// TIA Portal V21 export
FUNCTION "DIG IP" : Void   // FC3, LAD
{ S7_Optimized_Access := 'TRUE' }
// stored: SetENOAutomatically false
   VAR_TEMP   // added for the SCL form of the ladder/FBD networks
      _w1 : Bool;
      _w2 : Bool;
      _w3 : Bool;
      _w4 : Bool;
      _w5 : Bool;
   END_VAR
BEGIN

REGION Network 1: BLOCK CALL
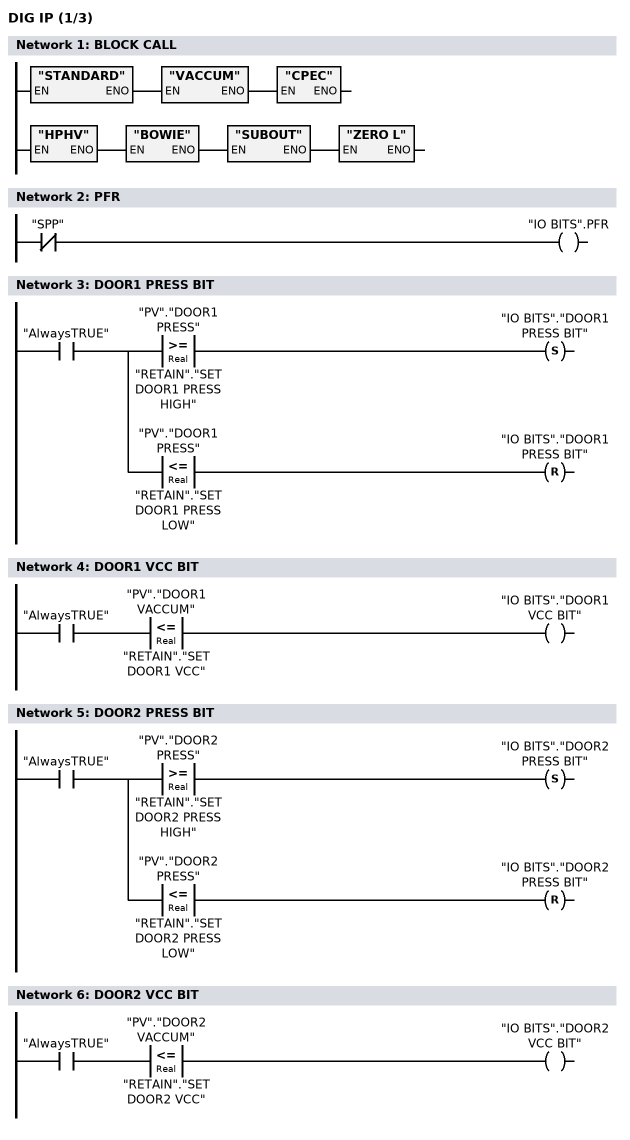
   RUNG wire#powerrail
      "STANDARD"()
      "VACCUM"()
      "CPEC"()
   END_RUNG
   RUNG wire#powerrail
      "HPHV"()
      "BOWIE"()
      "SUBOUT"()
      "ZERO L"()
   END_RUNG
   // the same network as SCL:
   "STANDARD"(ENO => #_w1);
   "VACCUM"(EN := #_w1, ENO => #_w2);
   IF #_w2 THEN "CPEC"(); END_IF;
   "HPHV"(ENO => #_w3);
   "BOWIE"(EN := #_w3, ENO => #_w4);
   "SUBOUT"(EN := #_w4, ENO => #_w5);
   IF #_w5 THEN "ZERO L"(); END_IF;
END_REGION

REGION Network 2: PFR
   RUNG wire#powerrail
      I_Contact( "SPP" )
      Coil( "IO BITS".PFR )
   END_RUNG
   // the same network as SCL:
   "IO BITS".PFR := NOT "SPP";
END_REGION

REGION Network 3: DOOR1 PRESS BIT
   RUNG wire#powerrail
      Contact( "AlwaysTRUE" )
      wire#w1
      { S7_Templates := "SrcType := Real" } GE_Contact(in1 := "PV"."DOOR1 PRESS", in2 := "RETAIN"."SET DOOR1 PRESS HIGH")
      S_Coil( "IO BITS"."DOOR1 PRESS BIT" )
   END_RUNG
   RUNG wire#w1
      { S7_Templates := "SrcType := Real" } LE_Contact(in1 := "PV"."DOOR1 PRESS", in2 := "RETAIN"."SET DOOR1 PRESS LOW")
      R_Coil( "IO BITS"."DOOR1 PRESS BIT" )
   END_RUNG
   // the same network as SCL:
   IF "AlwaysTRUE" AND ("PV"."DOOR1 PRESS" >= "RETAIN"."SET DOOR1 PRESS HIGH") THEN
       "IO BITS"."DOOR1 PRESS BIT" := TRUE;
   END_IF;
   IF "AlwaysTRUE" AND ("PV"."DOOR1 PRESS" <= "RETAIN"."SET DOOR1 PRESS LOW") THEN
       "IO BITS"."DOOR1 PRESS BIT" := FALSE;
   END_IF;
END_REGION

REGION Network 4: DOOR1 VCC BIT
   RUNG wire#powerrail
      Contact( "AlwaysTRUE" )
      { S7_Templates := "SrcType := Real" } LE_Contact(in1 := "PV"."DOOR1 VACCUM", in2 := "RETAIN"."SET DOOR1 VCC")
      Coil( "IO BITS"."DOOR1 VCC BIT" )
   END_RUNG
   // the same network as SCL:
   "IO BITS"."DOOR1 VCC BIT" := "AlwaysTRUE" AND ("PV"."DOOR1 VACCUM" <= "RETAIN"."SET DOOR1 VCC");
END_REGION

REGION Network 5: DOOR2 PRESS BIT
   RUNG wire#powerrail
      Contact( "AlwaysTRUE" )
      wire#w1
      { S7_Templates := "SrcType := Real" } GE_Contact(in1 := "PV"."DOOR2 PRESS", in2 := "RETAIN"."SET DOOR2 PRESS HIGH")
      S_Coil( "IO BITS"."DOOR2 PRESS BIT" )
   END_RUNG
   RUNG wire#w1
      { S7_Templates := "SrcType := Real" } LE_Contact(in1 := "PV"."DOOR2 PRESS", in2 := "RETAIN"."SET DOOR2 PRESS LOW")
      R_Coil( "IO BITS"."DOOR2 PRESS BIT" )
   END_RUNG
   // the same network as SCL:
   IF "AlwaysTRUE" AND ("PV"."DOOR2 PRESS" >= "RETAIN"."SET DOOR2 PRESS HIGH") THEN
       "IO BITS"."DOOR2 PRESS BIT" := TRUE;
   END_IF;
   IF "AlwaysTRUE" AND ("PV"."DOOR2 PRESS" <= "RETAIN"."SET DOOR2 PRESS LOW") THEN
       "IO BITS"."DOOR2 PRESS BIT" := FALSE;
   END_IF;
END_REGION

REGION Network 6: DOOR2 VCC BIT
   RUNG wire#powerrail
      Contact( "AlwaysTRUE" )
      { S7_Templates := "SrcType := Real" } LE_Contact(in1 := "PV"."DOOR2 VACCUM", in2 := "RETAIN"."SET DOOR2 VCC")
      Coil( "IO BITS"."DOOR2 VCC BIT" )
   END_RUNG
   // the same network as SCL:
   "IO BITS"."DOOR2 VCC BIT" := "AlwaysTRUE" AND ("PV"."DOOR2 VACCUM" <= "RETAIN"."SET DOOR2 VCC");
END_REGION

REGION Network 7: JACKET SAFETY BIT
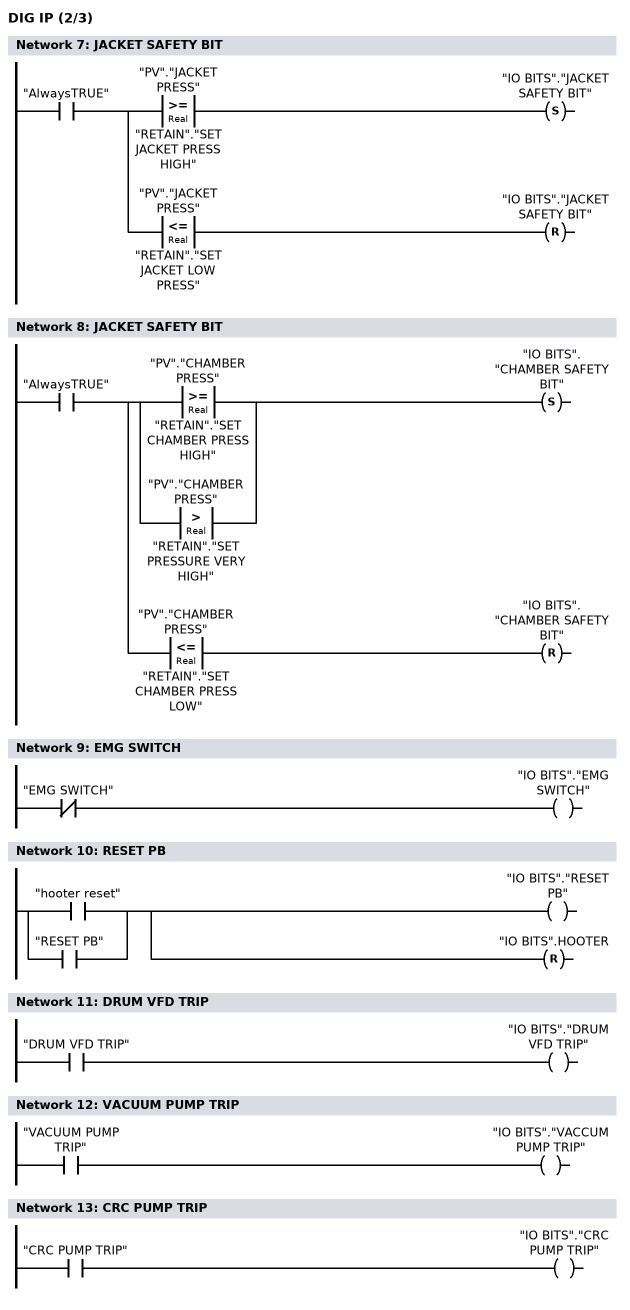
   RUNG wire#powerrail
      Contact( "AlwaysTRUE" )
      wire#w1
      { S7_Templates := "SrcType := Real" } GE_Contact(in1 := "PV"."JACKET PRESS", in2 := "RETAIN"."SET JACKET PRESS HIGH")
      S_Coil( "IO BITS"."JACKET SAFETY BIT" )
   END_RUNG
   RUNG wire#w1
      { S7_Templates := "SrcType := Real" } LE_Contact(in1 := "PV"."JACKET PRESS", in2 := "RETAIN"."SET JACKET LOW PRESS")
      R_Coil( "IO BITS"."JACKET SAFETY BIT" )
   END_RUNG
   // the same network as SCL:
   IF "AlwaysTRUE" AND ("PV"."JACKET PRESS" >= "RETAIN"."SET JACKET PRESS HIGH") THEN
       "IO BITS"."JACKET SAFETY BIT" := TRUE;
   END_IF;
   IF "AlwaysTRUE" AND ("PV"."JACKET PRESS" <= "RETAIN"."SET JACKET LOW PRESS") THEN
       "IO BITS"."JACKET SAFETY BIT" := FALSE;
   END_IF;
END_REGION

REGION Network 8: JACKET SAFETY BIT
   RUNG wire#powerrail
      Contact( "AlwaysTRUE" )
      wire#w1
      { S7_Templates := "SrcType := Real" } GE_Contact(in1 := "PV"."CHAMBER PRESS", in2 := "RETAIN"."SET CHAMBER PRESS HIGH")
      wire#w2
      S_Coil( "IO BITS"."CHAMBER SAFETY BIT" )
   END_RUNG
   RUNG wire#w1
      { S7_Templates := "SrcType := Real" } GT_Contact(in1 := "PV"."CHAMBER PRESS", in2 := "RETAIN"."SET PRESSURE VERY HIGH")
   END_RUNG wire#w2
   RUNG wire#w1
      { S7_Templates := "SrcType := Real" } LE_Contact(in1 := "PV"."CHAMBER PRESS", in2 := "RETAIN"."SET CHAMBER PRESS LOW")
      R_Coil( "IO BITS"."CHAMBER SAFETY BIT" )
   END_RUNG
   // the same network as SCL:
   IF "AlwaysTRUE" AND (("PV"."CHAMBER PRESS" >= "RETAIN"."SET CHAMBER PRESS HIGH") OR ("PV"."CHAMBER PRESS" > "RETAIN"."SET PRESSURE VERY HIGH")) THEN
       "IO BITS"."CHAMBER SAFETY BIT" := TRUE;
   END_IF;
   IF "AlwaysTRUE" AND ("PV"."CHAMBER PRESS" <= "RETAIN"."SET CHAMBER PRESS LOW") THEN
       "IO BITS"."CHAMBER SAFETY BIT" := FALSE;
   END_IF;
END_REGION

REGION Network 9: EMG SWITCH
   RUNG wire#powerrail
      I_Contact( "EMG SWITCH" )
      Coil( "IO BITS"."EMG SWITCH" )
   END_RUNG
   // the same network as SCL:
   "IO BITS"."EMG SWITCH" := NOT "EMG SWITCH";
END_REGION

REGION Network 10: RESET PB
   RUNG wire#powerrail
      Contact( "hooter reset" )
      wire#w1
      Coil( "IO BITS"."RESET PB" )
   END_RUNG
   RUNG wire#powerrail
      Contact( "RESET PB" )
   END_RUNG wire#w1
   RUNG wire#w1
      R_Coil( "IO BITS".HOOTER )
   END_RUNG
   // the same network as SCL:
   "IO BITS"."RESET PB" := "hooter reset" OR "RESET PB";
   IF "IO BITS"."RESET PB" THEN "IO BITS".HOOTER := FALSE; END_IF;
END_REGION

REGION Network 11: DRUM VFD TRIP
   RUNG wire#powerrail
      Contact( "DRUM VFD TRIP" )
      Coil( "IO BITS"."DRUM VFD TRIP" )
   END_RUNG
   // the same network as SCL:
   "IO BITS"."DRUM VFD TRIP" := "DRUM VFD TRIP";
END_REGION

REGION Network 12: VACUUM PUMP TRIP
   RUNG wire#powerrail
      Contact( "VACUUM PUMP TRIP" )
      Coil( "IO BITS"."VACCUM PUMP TRIP" )
   END_RUNG
   // the same network as SCL:
   "IO BITS"."VACCUM PUMP TRIP" := "VACUUM PUMP TRIP";
END_REGION

REGION Network 13: CRC PUMP TRIP
   RUNG wire#powerrail
      Contact( "CRC PUMP TRIP" )
      Coil( "IO BITS"."CRC PUMP TRIP" )
   END_RUNG
   // the same network as SCL:
   "IO BITS"."CRC PUMP TRIP" := "CRC PUMP TRIP";
END_REGION

REGION Network 14: DOOR1 OPEN LMT
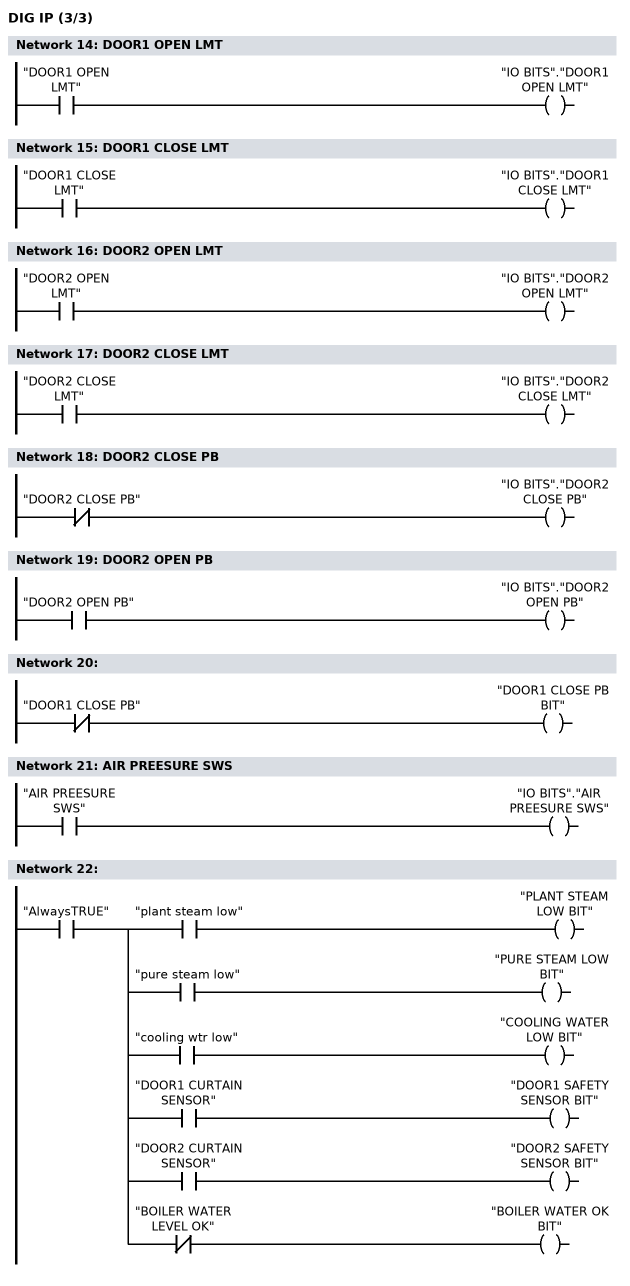
   RUNG wire#powerrail
      Contact( "DOOR1 OPEN LMT" )
      Coil( "IO BITS"."DOOR1 OPEN LMT" )
   END_RUNG
   // the same network as SCL:
   "IO BITS"."DOOR1 OPEN LMT" := "DOOR1 OPEN LMT";
END_REGION

REGION Network 15: DOOR1 CLOSE LMT
   RUNG wire#powerrail
      Contact( "DOOR1 CLOSE LMT" )
      Coil( "IO BITS"."DOOR1 CLOSE LMT" )
   END_RUNG
   // the same network as SCL:
   "IO BITS"."DOOR1 CLOSE LMT" := "DOOR1 CLOSE LMT";
END_REGION

REGION Network 16: DOOR2 OPEN LMT
   RUNG wire#powerrail
      Contact( "DOOR2 OPEN LMT" )
      Coil( "IO BITS"."DOOR2 OPEN LMT" )
   END_RUNG
   // the same network as SCL:
   "IO BITS"."DOOR2 OPEN LMT" := "DOOR2 OPEN LMT";
END_REGION

REGION Network 17: DOOR2 CLOSE LMT
   RUNG wire#powerrail
      Contact( "DOOR2 CLOSE LMT" )
      Coil( "IO BITS"."DOOR2 CLOSE LMT" )
   END_RUNG
   // the same network as SCL:
   "IO BITS"."DOOR2 CLOSE LMT" := "DOOR2 CLOSE LMT";
END_REGION

REGION Network 18: DOOR2 CLOSE PB
   RUNG wire#powerrail
      I_Contact( "DOOR2 CLOSE PB" )
      Coil( "IO BITS"."DOOR2 CLOSE PB" )
   END_RUNG
   // the same network as SCL:
   "IO BITS"."DOOR2 CLOSE PB" := NOT "DOOR2 CLOSE PB";
END_REGION

REGION Network 19: DOOR2 OPEN PB
   RUNG wire#powerrail
      Contact( "DOOR2 OPEN PB" )
      Coil( "IO BITS"."DOOR2 OPEN PB" )
   END_RUNG
   // the same network as SCL:
   "IO BITS"."DOOR2 OPEN PB" := "DOOR2 OPEN PB";
END_REGION

REGION Network 20
   RUNG wire#powerrail
      I_Contact( "DOOR1 CLOSE PB" )
      Coil( "DOOR1 CLOSE PB BIT" )
   END_RUNG
   // the same network as SCL:
   "DOOR1 CLOSE PB BIT" := NOT "DOOR1 CLOSE PB";
END_REGION

REGION Network 21: AIR PREESURE SWS
   RUNG wire#powerrail
      Contact( "AIR PREESURE SWS" )
      Coil( "IO BITS"."AIR PREESURE SWS" )
   END_RUNG
   // the same network as SCL:
   "IO BITS"."AIR PREESURE SWS" := "AIR PREESURE SWS";
END_REGION

REGION Network 22
   RUNG wire#powerrail
      Contact( "AlwaysTRUE" )
      wire#w1
      Contact( "plant steam low" )
      Coil( "PLANT STEAM LOW BIT" )
   END_RUNG
   RUNG wire#w1
      Contact( "pure steam low" )
      Coil( "PURE STEAM LOW BIT" )
   END_RUNG
   RUNG wire#w1
      Contact( "cooling wtr low" )
      Coil( "COOLING WATER LOW BIT" )
   END_RUNG
   RUNG wire#w1
      Contact( "DOOR1 CURTAIN SENSOR" )
      Coil( "DOOR1 SAFETY SENSOR BIT" )
   END_RUNG
   RUNG wire#w1
      Contact( "DOOR2 CURTAIN SENSOR" )
      Coil( "DOOR2 SAFETY SENSOR BIT" )
   END_RUNG
   RUNG wire#w1
      I_Contact( "BOILER WATER LEVEL OK" )
      Coil( "BOILER WATER OK BIT" )
   END_RUNG
   // the same network as SCL:
   "PLANT STEAM LOW BIT" := "AlwaysTRUE" AND "plant steam low";
   "PURE STEAM LOW BIT" := "AlwaysTRUE" AND "pure steam low";
   "COOLING WATER LOW BIT" := "AlwaysTRUE" AND "cooling wtr low";
   "DOOR1 SAFETY SENSOR BIT" := "AlwaysTRUE" AND "DOOR1 CURTAIN SENSOR";
   "DOOR2 SAFETY SENSOR BIT" := "AlwaysTRUE" AND "DOOR2 CURTAIN SENSOR";
   "BOILER WATER OK BIT" := "AlwaysTRUE" AND NOT "BOILER WATER LEVEL OK";
END_REGION
END_FUNCTION
